Fanuc KAREL source: kb00083.KL

-- PROVISIONAL review KL for V940-1; original PC SHA256 f5eb5ec0e9258d8ec8807c30943118c59d19a95b4bc5037444285eece60f6edf
-- Incomplete behavior may be omitted. Consult companion uncertainty JSON. Do not deploy.
PROGRAM KB00083
%NOLOCKGROUP
BEGIN
  -- V9_ZERO_TABLE_METADATA_HINT layout=0002_ascii; no indexed target words; source/name/runtime held
  -- UNRESOLVED_PC offsets 5-12; opcodes 9D,23
  -- UNRESOLVED_PC offsets 17-24; opcodes 9D,23
  -- UNRESOLVED_PC offsets 29-36; opcodes 9D,23
  -- UNRESOLVED_PC offsets 41-48; opcodes 9D,23
  -- UNRESOLVED_PC offsets 53-81; opcodes 27,22,22,22,22,31
  -- UNRESOLVED_PC offsets 86-90; opcodes 7F
END KB00083
